FUNCTION_BLOCK ExitCheck (* Template for a Basic Function Block Type *)
  (* Standard: 61499-2 *)
  (* Version 1.0, 2021-07-29, Tuojian Lyu *)
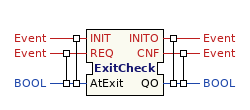
  EVENT_INPUT
    INIT WITH AtExit; (* Initialization Request *)
    REQ WITH AtExit; (* Normal Execution Request *)
  END_EVENT
  EVENT_OUTPUT
    INITO WITH QO; (* Initialization Confirm *)
    CNF WITH QO; (* Execution Confirmation *)
  END_EVENT
  VAR_INPUT
    AtExit : BOOL; (* Input event qualifier *)
  END_VAR
  VAR_OUTPUT
    QO : BOOL; (* Output event qualifier *)
  END_VAR
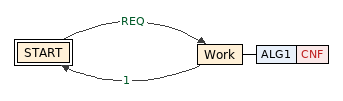
  EC_STATES
    START; (* Initial State *)
    Work : ALG1 -> CNF;
  END_STATES
  EC_TRANSITIONS
    START TO Work := REQ;
    Work TO START := 1;
  END_TRANSITIONS
  ALGORITHM ALG1 IN ST:
IF (TRUE = AtExit) THEN
QO := TRUE;
END_IF;
  END_ALGORITHM
END_FUNCTION_BLOCK
